// TIA Portal V16 export
// export: Created 2024-09-05T17:40:15.0323535Z, ExportSetting WithDefaults, DisplayName Totally Integrated Automation Portal, DisplayVersion V16 Update 6, DisplayName TIA Portal Version Control Interface, DisplayVersion V16 Update 2, DisplayName TIA Portal Openness, DisplayVersion V16 Update 6, DisplayName STEP 7 Professional, DisplayVersion V16 Update 6, DisplayName STEP 7 Safety, DisplayVersion V16, DisplayName WinCC Advanced, DisplayVersion V16 Update 6
TYPE "UDT_HydraulicCylinderData"
// stored: IsFailsafeCompliant false
   STRUCT
      Pressure : Real;
      Flow : Real;
      Position : Real;
      StandstillPosition : Real;
      PressureCmd : Real;
      FlowCmd : Real;
      PressureBack : Real;
      FlowBack : Real;
      HAxis : Real;
      Force : Real;
      Status : "UDT_Cylinder";
      InBp_1mm_margin { S7_SetPoint := 'True'} : Bool;
   END_STRUCT;
END_TYPE
